FUNCTION Fill_Row_Four : BOOL
VAR_INPUT
	row: ARRAY[1..10] OF WORD;
END_VAR
VAR
END_VAR

GV_MODBUS.fourLeft[1]:= row[1];
GV_MODBUS.fourLeft[2]:= row[2];
GV_MODBUS.fourLeft[3]:= row[3];
GV_MODBUS.fourLeft[4]:= row[4];
GV_MODBUS.fourLeft[5]:= row[5];
GV_MODBUS.fourRight[1]:= row[6];
GV_MODBUS.fourRight[2]:= row[7];
GV_MODBUS.fourRight[3]:= row[8];
GV_MODBUS.fourRight[4]:= row[9];
GV_MODBUS.fourRight[5]:= row[10];

END_FUNCTION

(* stored: Version 1.1.0.1, ProductVersion 3.1.4022.12
   POU Fill_Row_Four: Id {b42078dc-a20e-4214-9910-ebf83dbff697}, SpecialFunc None *)
